TEXTLIST TextList_tabvac_errorid
  0 = 'no_error'
  1 = 'not_connected'
  2 = 'invalid_state'
  3 = 'vacuum_on_timeout'
  4 = 'vacuum_off_timeout'
  5 = 'cmd_timeout'
  6 = 'TBD_error'
  7 = 'io_error'
  8 = 'unknown_error'
  666 = 'emergency_error'
   = ''
END_TEXTLIST

(* stored: Version 1.1.0.1, ProductVersion 3.1.4024.11
   TextList TextList_tabvac_errorid: Id {ed53f633-b37e-409b-b73f-ae316064bebc} *)
